PROGRAM MAIN
VAR
	
	
	{attribute addProperty Name "<#Hello#> <#World#>"}
	Hello_World : STRING;
	
	{attribute wpf [RenderIgnore()]}
	progressBar: stProgressBar;
	
	stations : stStations;
	
END_VAR

Hello_World := 'This is automatically generated UI!' ;
IF progressBar.testBool = TRUE THEN
	progressBar.testInteger := progressBar.testInteger + 1;
	IF progressBar.testInteger = 1000 THEN
		progressBar.testBool := FALSE; 
	END_IF
END_IF

END_PROGRAM

(* stored: Version 1.1.0.1, ProductVersion 3.1.4024.6
   POU MAIN: Id {2aec7386-fec2-4299-8c2e-88bb20ee3274}, SpecialFunc None *)
